(* IEC 61131-3 sources: PLC_MixingTank/StorageTank/FB, 4 files *)

(* ---- FB_TankLevelSim_Var.st ---- *)
FUNCTION_BLOCK FB_TankLevelSim
VAR_INPUT
    XOValveActive : BOOL;
    DrainValveActive : BOOL;
    DischargeValveActive : BOOL;

    XOFillRate : REAL := 8.0;
    DrainRate : REAL := 15.0;
    DischargeRate : REAL := 3.0;

    Execute : BOOL;
    Reset : BOOL;
    InitialLevel : REAL := 0.0;
END_VAR

VAR_OUTPUT
    SimulatedLevel : REAL := 0.0;
END_VAR

VAR
    RawTrig : R_TRIG;
    dLevel : REAL;
END_VAR

(* ---- FB_TankTempSim_Var.st ---- *)
FUNCTION_BLOCK FB_TankTempSim
VAR_INPUT
    SteamValveInput : REAL;

    Execute : BOOL;
    Reset : BOOL;

    MaxHeatingPerSec : REAL := 0.05;
    AmbientTemp : REAL := 25.0;
    HeatLossCoeff : REAL := 0.001;
END_VAR

VAR_OUTPUT
    SimulatedTemp : REAL := 25.0;
END_VAR

VAR
    dTemp : REAL;
END_VAR

(* ---- FB_PID_Exe.st ---- *)
IF NOT Enable THEN
    Integral := 0.0;
    PrevError := 0.0;
    Out := 0.0;
    Error := 0.0;
ELSE
    Error := SetPoint - ProcessValue;

    IF Ti > 0.0 AND CycleTime > 0.0 THEN
        Integral := Integral + ((CycleTime * Error) / Ti);
    ELSE
        Integral := 0.0;
    END_IF

    IF CycleTime > 0.0 THEN
        Derivative := (Error - PrevError) / CycleTime * Td;
    ELSE
        Derivative := 0.0;
    END_IF

    RawOut := Kp * (Error + Integral + Derivative);

    IF RawOut > OutMax THEN
        Out := OutMax;
        IF Ti > 0.0  AND CycleTime > 0.0 THEN
            Integral := Integral - ((CycleTime * Error) / Ti);
        END_IF
    ELSIF RawOut < OutMin THEN
        Out := OutMin;
        IF Ti > 0.0 AND CycleTime > 0.0 THEN
            Integral := Integral - ((CycleTime * Error)/ Ti);
        END_IF
    ELSE
        Out := RawOut;
    END_IF
    PrevError := Error;
END_IF

(* ---- FB_TankLevelSim_Exe.st ---- *)
IF Reset THEN
    SimulatedLevel := InitialLevel;
ELSIF Execute THEN
    dLevel := 0.0;

    IF XOValveActive THEN
        dLevel := dLevel + XOFillRate;
    END_IF

    IF DischargeValveActive THEN
        dLevel := dLevel - DischargeRate;
    END_IF

    IF DrainValveActive THEN
        dLevel := dLevel - DrainRate;
    END_IF

    SimulatedLevel := SimulatedLevel + dLevel;

    IF SimulatedLevel < 0.0 THEN
        SimulatedLevel := 0.0;
    END_IF
END_IF
